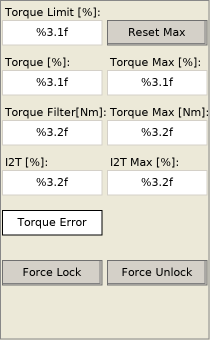
VISUALIZATION PH_Motor  // 210x340
//==================================================================================================
//							Beckhoff Automation Poland
//									18.04.2018
//	Wizualizacja dla Axis Online
//  v1.0	|| TC v 3.1.4022.16		|| - pierwsza wersja
//==================================================================================================
VAR_IN_OUT
	stMcAxisOnline			: ST_McAxisOnline;	
END_VAR
    Button (107,20 100x25), "Reset Max"
        tap stMcAxisOnline.stMotorMonitoring.bReset
    Group (2,0 100x45)
        Textfield (0,20 100x25), "%3.1f", text variable: stMcAxisOnline.stMotorMonitoring.rTorqueLimit
            OnMouseClick: write the text variable via InputWithLimits, min 0, max 500
        Label (0,0 100x25), "Torque Limit [%]:"
    Rectangle (2,210 100x25), "Torque Error", colour toggle: stMcAxisOnline.stMotorMonitoring.bError
    Group (2,100 100x45)
        Textfield (0,20 100x25), "%3.2f", text variable: stMcAxisOnline.stMotorMonitoring.rTorqueF, colour toggle: stMcAxisOnline.stMotorMonitoring.bWarning
        Label (0,0 100x25), "Torque Filter[Nm]:"
    Group (107,100 100x45)
        Textfield (0,20 100x25), "%3.2f", text variable: stMcAxisOnline.stMotorMonitoring.rTorqueMax
        Label (0,0 100x25), "Torque Max [Nm]:"
    Group (2,150 100x45)
        Label (0,0 100x25), "I2T [%]:"
        Textfield (0,20 100x25), "%3.2f", text variable: stMcAxisOnline.stMotorMonitoring.rI2T
    Group (107,150 100x45)
        Label (0,0 100x25), "I2T Max [%]:"
        Textfield (0,20 100x25), "%3.2f", text variable: stMcAxisOnline.stMotorMonitoring.rI2TMax
    Button (2,260 100x25), "Force Lock"
        tap stMcAxisOnline.stHoldingBrake.bForceLock
    Button (107,260 100x25), "Force Unlock"
        tap stMcAxisOnline.stHoldingBrake.bForceUnlock
    Group (2,50 100x45)
        Textfield (0,20 100x25), "%3.1f", text variable: stMcAxisOnline.stMotorMonitoring.rTorquePerc, colour toggle: stMcAxisOnline.stMotorMonitoring.bWarning
        Label (0,0 100x25), "Torque [%]:"
    Group (107,50 100x45)
        Textfield (0,20 100x25), "%3.1f", text variable: stMcAxisOnline.stMotorMonitoring.rTorquePercMax
        Label (0,0 100x25), "Torque Max [%]:"
END_VISUALIZATION

(* stored: Version 1.1.0.1, ProductVersion 3.1.4022.10
   Visu PH_Motor: Id {97d15dbc-fcaf-4255-982b-0fdd32e9d896} *)
